(* PLC project PLC, Beckhoff Automation GmbH TwinCAT PLC Control 3.5.13.21 *)
(* stored: creationDateTime 2024-02-17T22:42:45.2426081, modificationDateTime 2024-02-17T22:42:45.2426081 *)

TYPE CylConfig :
STRUCT
	operateDelayTime: TIME;
	sensorDelayTime: TIME;
	cylinderErrorTime: TIME;
END_STRUCT
END_TYPE
